(* IEC 61131-3 sources: repolevel_ST_code_completion/real_groud_truth最新/repoeval_plc_hello_mixing_tank/readful_result, 6 files *)

(* ---- FB_AutoSequence.st ---- *)
VAR
	// 内部状态变量
	eNextState			:	AUTO_SEQUENCE;	// 下一个状态
	tStateTimer			:	TIME;			// 状态计时器
	nCycleCounter		:	UINT := 0;		// 循环计数器
	bTransitionFlag		:	BOOL := FALSE;	// 状态转换标志
END_VAR

// 自动序列状态枚举
TYPE AUTO_SEQUENCE :
(
	IDLE,				// 空闲状态
	FILLING_MEDIUM1,	// 介质1填充状态
	FILLING_MEDIUM2,	// 介质2填充状态
	MIXING,				// 混合状态
	DRAINING			// 排空状态
);
END_TYPE

// 自动序列逻辑实现
IF bEnable THEN
	CASE eCurrentState OF
		IDLE:
			IF bTankLevelEmpty THEN
				eNextState := FILLING_MEDIUM1;
			END_IF;

		FILLING_MEDIUM1:
			bMedium1OpenCmd := TRUE;
			IF bTankLevelFull THEN
				bMedium1OpenCmd := FALSE;
				eNextState := FILLING_MEDIUM2;
			END_IF;

		FILLING_MEDIUM2:
			bMedium2OpenCmd := TRUE;
			IF bTankLevelFull THEN
				bMedium2OpenCmd := FALSE;
				eNextState := MIXING;
			END_IF;

		MIXING:
			bMixerRunCmd := TRUE;
			IF tStateTimer >= tMixingDuration THEN
				bMixerRunCmd := FALSE;
				eNextState := DRAINING;
			END_IF;

		DRAINING:
			bDrainOpenCmd := TRUE;
			IF bTankLevelEmpty THEN
				bDrainOpenCmd := FALSE;
				eNextState := IDLE;
				nCycleCounter := nCycleCounter + 1;
			END_IF;
	END_CASE;

	// 状态更新
	IF eNextState <> eCurrentState THEN
		eCurrentState := eNextState;
		tStateTimer := T#0S; // 重置状态计时器
	END_IF;

	// 状态计时器更新
	tStateTimer := tStateTimer + T#1MS;
ELSE
	// 禁用时复位所有命令和状态
	bMixerRunCmd := FALSE;
	bMedium1OpenCmd := FALSE;
	bMedium2OpenCmd := FALSE;
	bDrainOpenCmd := FALSE;
	eCurrentState := IDLE;
	nCycleCounter := 0;
END_IF;

IF bReset THEN
	// 复位逻辑
	bMixerRunCmd := FALSE;
	bMedium1OpenCmd := FALSE;
	bMedium2OpenCmd := FALSE;
	bDrainOpenCmd := FALSE;
	eCurrentState := IDLE;
	nCycleCounter := 0;
	tStateTimer := T#0S;
END_IF;

(* ---- FB_ModeController.st ---- *)
VAR
	ePreviousMode	:	MODES;	// 上一次模式
END_VAR

// 定义模式类型
TYPE MODES : (MANUAL, AUTO);
END_TYPE

// 初始化
IF NOT eCurrentMode THEN
	eCurrentMode := MANUAL; // 默认模式为手动模式
	ePreviousMode := MANUAL;
	bModeChanged := FALSE;
END_IF

// 模式切换逻辑
IF bSetToAuto AND (eCurrentMode <> AUTO) THEN
	ePreviousMode := eCurrentMode;
	eCurrentMode := AUTO;
	bModeChanged := TRUE;
ELSIF bSetToManual AND (eCurrentMode <> MANUAL) THEN
	ePreviousMode := eCurrentMode;
	eCurrentMode := MANUAL;
	bModeChanged := TRUE;
ELSE
	bModeChanged := FALSE;
END_IF

(* ---- F_ResetDeviceCommands.st ---- *)
VAR_OUTPUT
	// 复位完成标志
	bResetComplete		:	BOOL;
END_VAR

// 功能描述：复位所有HMI命令标志，当设备状态与命令一致时完成复位
bResetComplete := FALSE;

// 混合电机命令复位逻辑
IF NOT bMixerRunning AND bMixerRunCmd THEN
	bMixerRunCmd := FALSE;
END_IF;

IF bMixerRunning AND bMixerStopCmd THEN
	bMixerStopCmd := FALSE;
END_IF;

// Medium1命令复位逻辑
IF NOT bMedium1Opened AND bMedium1OpenCmd THEN
	bMedium1OpenCmd := FALSE;
END_IF;

IF bMedium1Opened AND bMedium1CloseCmd THEN
	bMedium1CloseCmd := FALSE;
END_IF;

// Medium2命令复位逻辑
IF NOT bMedium2Opened AND bMedium2OpenCmd THEN
	bMedium2OpenCmd := FALSE;
END_IF;

IF bMedium2Opened AND bMedium2CloseCmd THEN
	bMedium2CloseCmd := FALSE;
END_IF;

// Drain命令复位逻辑
IF NOT bDrainOpened AND bDrainOpenCmd THEN
	bDrainOpenCmd := FALSE;
END_IF;

IF bDrainOpened AND bDrainCloseCmd THEN
	bDrainCloseCmd := FALSE;
END_IF;

// 检查是否所有命令标志已复位
IF NOT bMixerRunCmd AND NOT bMixerStopCmd AND
   NOT bMedium1OpenCmd AND NOT bMedium1CloseCmd AND
   NOT bMedium2OpenCmd AND NOT bMedium2CloseCmd AND
   NOT bDrainOpenCmd AND NOT bDrainCloseCmd THEN
	bResetComplete := TRUE;
END_IF;

RETURN bResetComplete;
END_FUNCTION

(* ---- F_UpdateLimitSwitches.st ---- *)
# --------------------------------------------------
# FUNCTION F_UpdateLimitSwitches
# This function updates the limit switches based on the current tank level.
# If the tank level exceeds the full threshold, the full switch is activated.
# If the tank level drops below the empty threshold, the empty switch is activated.
# --------------------------------------------------

# Update the full level switch
IF rTankLevel >= rFullThreshold THEN
    bLevelFull := TRUE;
ELSE
    bLevelFull := FALSE;
END_IF;

# Update the empty level switch
IF rTankLevel <= rEmptyThreshold THEN
    bLevelEmpty := TRUE;
ELSE
    bLevelEmpty := FALSE;
END_IF;

# Return TRUE to indicate the function executed successfully
F_UpdateLimitSwitches := TRUE;

(* ---- FB_ManualControl.st ---- *)
VAR
	// 内部变量
	bResetCommands		:	BOOL;
END_VAR

// 主程序逻辑
// 复位命令逻辑
bResetCommands := F_ResetDeviceCommands(
	bMixerRunCmd := bMixerRunCmd,
	bMixerStopCmd := bMixerStopCmd,
	bMedium1OpenCmd := bMedium1OpenCmd,
	bMedium1CloseCmd := bMedium1CloseCmd,
	bMedium2OpenCmd := bMedium2OpenCmd,
	bMedium2CloseCmd := bMedium2CloseCmd,
	bDrainOpenCmd := bDrainOpenCmd,
	bDrainCloseCmd := bDrainCloseCmd,
	bMixerRunning := bMixerRunning,
	bMedium1Opened := bMedium1Opened,
	bMedium2Opened := bMedium2Opened,
	bDrainOpened := bDrainOpened
);

// 输出命令逻辑
IF bMixerRunCmd AND NOT bMixerRunning THEN
	bMixerRunCmdOut := TRUE;	// 启动混合电机
ELSE
	bMixerRunCmdOut := FALSE;
END_IF

IF bMedium1OpenCmd AND NOT bMedium1Opened THEN
	bMedium1OpenCmdOut := TRUE;	// 打开介质1阀门
ELSE
	bMedium1OpenCmdOut := FALSE;
END_IF

IF bMedium2OpenCmd AND NOT bMedium2Opened THEN
	bMedium2OpenCmdOut := TRUE;	// 打开介质2阀门
ELSE
	bMedium2OpenCmdOut := FALSE;
END_IF

IF bDrainOpenCmd AND NOT bDrainOpened THEN
	bDrainOpenCmdOut := TRUE;	// 打开排空阀门
ELSE
	bDrainOpenCmdOut := FALSE;
END_IF

(* ---- FB_TankLevelSimulator.st ---- *)
VAR
	rLevel				:	REAL;			// 内部液位变量
END_VAR

// 初始化液位
IF bReset THEN
	rLevel := rInitialLevel;
END_IF

// 液位计算逻辑
IF bMedium1Opened THEN
	rLevel := rLevel + rFillRate1;
END_IF

IF bMedium2Opened THEN
	rLevel := rLevel + rFillRate2;
END_IF

IF bDrainOpened THEN
	rLevel := rLevel - rDrainRate;
END_IF

// 限制液位范围
IF rLevel < rMinLevel THEN
	rLevel := rMinLevel;
ELSIF rLevel > rMaxLevel THEN
	rLevel := rMaxLevel;
END_IF

// 输出当前液位
rCurrentLevel := rLevel;
